FUNCTION_BLOCK Robot (* Template for a simple Basic Function Block Type *)
  (* Standard: 61499-2 *)
  (* Version 1.0, 2019-04-03, michael *)
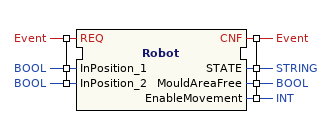
  EVENT_INPUT
    REQ WITH InPosition_1, InPosition_2; (* Initialization Request *)
  END_EVENT
  EVENT_OUTPUT
    CNF WITH MouldAreaFree, EnableMovement, STATE; (* Execution Confirmation *)
  END_EVENT
  VAR_INPUT
    InPosition_1 : BOOL; (* Mould Closed *)
    InPosition_2 : BOOL; (* Mould Opened *)
  END_VAR
  VAR_OUTPUT
    STATE : STRING;
    MouldAreaFree : BOOL := FALSE; (* Output event qualifier *)
    EnableMovement : INT := 3;
  END_VAR
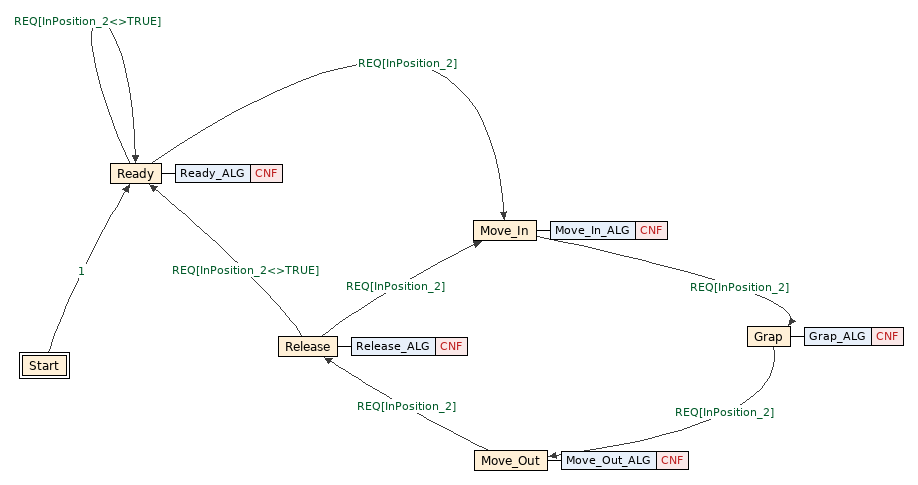
  EC_STATES
    Start; (* Initial State *)
    Move_In : Move_In_ALG -> CNF;
    Grap : Grap_ALG -> CNF;
    Move_Out : Move_Out_ALG -> CNF;
    Release : Release_ALG -> CNF;
    Ready : Ready_ALG -> CNF;
  END_STATES
  EC_TRANSITIONS
    Move_In TO Grap := REQ[InPosition_2];
    Grap TO Move_Out := REQ[InPosition_2];
    Release TO Move_In := REQ[InPosition_2];
    Move_Out TO Release := REQ[InPosition_2];
    Release TO Ready := REQ[InPosition_2<>TRUE];
    Ready TO Move_In := REQ[InPosition_2];
    Start TO Ready := 1;
    Ready TO Ready := REQ[InPosition_2<>TRUE];
  END_TRANSITIONS
  ALGORITHM Move_In_ALG IN ST: (* new algorithm *)
STATE:="MOVE_IN";
MouldAreaFree:=FALSE;
EnableMovement:=1;
  END_ALGORITHM
  ALGORITHM Move_Out_ALG IN ST: (* new algorithm *)
STATE:="MOVE_OUT";
MouldAreaFree:=TRUE;
EnableMovement:=3;
  END_ALGORITHM
  ALGORITHM Grap_ALG IN ST: (* new algorithm *)
STATE:="GRAP";
MouldAreaFree:=FALSE;
EnableMovement:=1;
  END_ALGORITHM
  ALGORITHM Release_ALG IN ST: (* new algorithm *)
STATE:="Release";
MouldAreaFree:=TRUE;
EnableMovement:=3;
  END_ALGORITHM
  ALGORITHM Ready_ALG IN ST: (* new algorithm *)
STATE:="Ready";
MouldAreaFree:=TRUE;
EnableMovement:=0;
  END_ALGORITHM
END_FUNCTION_BLOCK
